{attribute 'GeneratedUsingTerminal: EJ9576-0000-0018'}
{attribute addProperty BoxType "EJ9576-0000-0018"}
{attribute addProperty Id "EtcSlaveTerminalBaseBCT_InputsAT %I*BCT_Inputs_8E55234D16WcStateAT %I*WcState_9091E0EB2InfoDataAT %I*InfoData_32EB74EA10"}
{attribute addProperty CRC "1868358691"}
{attribute addProperty Size "28"}
TYPE EJ9576_6F5CE423 EXTENDS EtcSlaveTerminalBase :
STRUCT
	{attribute addProperty Name "BCT_Inputs"}
	BCT_Inputs : BCT_Inputs_8E55234D;
	{attribute addProperty Name "WcState"}
	WcState : WcState_9091E0EB;
	{attribute addProperty Name "InfoData"}
	InfoData : InfoData_32EB74EA;
END_STRUCT
END_TYPE

(* stored: Version 1.2.0.0, ProductVersion 3.1.4024.9
   DUT EJ9576_6F5CE423: Id {c934e373-e1e0-4ad5-a8f2-32da7ed2bdfa} *)
